INTERFACE I_MbTransport

METHOD Abort
VAR_INPUT
	nUnitId : USINT;
END_VAR
END_METHOD

METHOD Acquire : BOOL
VAR_INPUT
	nUnitId : USINT;   // Caller's unit ID doubles as the owner key. TRUE = you hold the bus.
END_VAR
END_METHOD

PROPERTY bReady : BOOL
GET
END_GET
END_PROPERTY

PROPERTY eLastError : E_MbErrorClass
GET
END_GET
END_PROPERTY

METHOD Poll : E_MbXferState
END_METHOD

PROPERTY pResponsePdu : POINTER TO BYTE
GET
END_GET
END_PROPERTY

PROPERTY PropcbResponsePdu : UINT
GET
END_GET
END_PROPERTY

METHOD Release
VAR_INPUT
	nUnitId : USINT;
END_VAR
END_METHOD

METHOD Send : BOOL
VAR_INPUT
	nUnitId         : USINT;
	pPdu            : POINTER TO BYTE;
	cbPdu           : UINT;
	nExpectedPduLen : UINT;   // From F_MbExpectedResponseLength; RTU uses it to detect end of frame
	tTimeout        : TIME;
END_VAR
END_METHOD

END_INTERFACE

(* stored: Version 1.1.0.1
   Itf I_MbTransport: Id {5e2641e3-5baf-4f56-8acb-08ba34d5721e}
   Method Abort: Id {a2414c33-193c-497e-91ff-055b80211172}
   Method Acquire: Id {e8b6dc96-6c1b-4695-bdcc-5ed702abeade}
   Property bReady: Id {f1f3f453-f257-4808-a9e5-352f0af6b022}
   Get Get: Id {7603ea32-7a8f-42e5-a6d3-5c31ca8e950d}
   Property eLastError: Id {12e97a06-a77c-47e6-8562-6ee6ecbb97d0}
   Get Get: Id {4e997a8d-5f67-4e7a-ac76-cb450b3b1cbf}
   Method Poll: Id {80eb6a04-8139-4b76-bdf6-a69ed141e4ca}
   Property pResponsePdu: Id {e153f7db-31a4-4089-88ee-fdf20448a932}
   Get Get: Id {81eb4523-6382-477e-8df0-67db6671c07d}
   Property PropcbResponsePdu: Id {814f7d24-46a3-4272-9512-7c132007175c}
   Get Get: Id {e18db762-d5ce-4f7a-aa92-8e2ae1e693e7}
   Method Release: Id {a55f0abe-f856-45ff-bf30-7d1d38b9d74e}
   Method Send: Id {a0027438-c754-4ef1-8b32-34073cc05afd} *)
